// TIA Portal project "XC221" (V12)

(* hardware
DEVICE "S7-1200 station_1"  SIMATIC 1200-Station
   slot 0: "S7-1200 rack"  Rack  V1.0
   slot 1: "PLC_123"  CPU 1214C DC/DC/DC  6ES7 214-1AG31-0XB0  V3.0
   slot 3: "AQ1 x 12 bits"  6ES7 232-4HA30-0XB0  V1.0
*)

// ===== PLC "PLC_123"  CPU 1214C DC/DC/DC =====
// protected blocks, not shown: "EASYPI", "MEMRST"

VAR_GLOBAL   // PLC tag table "Default tag table"
   "System_Byte" AT %MB1 : Byte;
   "FirstScan" AT %M1.0 : Bool;
   "DiagStatusUpdate" AT %M1.1 : Bool;
   "AlwaysTRUE" AT %M1.2 : Bool;
   "AlwaysFALSE" AT %M1.3 : Bool;
   "Clock_Byte" AT %MB0 : Byte;
   "Clock_10Hz" AT %M0.0 : Bool;
   "Clock_5Hz" AT %M0.1 : Bool;
   "Clock_2.5Hz" AT %M0.2 : Bool;
   "Clock_2Hz" AT %M0.3 : Bool;
   "Clock_1.25Hz" AT %M0.4 : Bool;
   "Clock_1Hz" AT %M0.5 : Bool;
   "Clock_0.625Hz" AT %M0.6 : Bool;
   "Clock_0.5Hz" AT %M0.7 : Bool;
END_VAR

VAR_GLOBAL   // PLC tag table "11 - Parâmetros"
   "Par_VT101_HorLim" AT %MD705 : Real;   // Limite de Horas do Ventilador 1
   "Par_VT102_HorLim" AT %MD709 : Real;   // Limite de Horas do Ventilador 2
   "Par_LT101_LimHH" AT %MD713 : Real;   // Limite para a condição “Muito Alto” [mm]
   "Par_LT101_LimH" AT %MD717 : Real;   // Limite para a condição “Alto” [mm]
   "Par_LT101_LimL" AT %MD721 : Real;   // Limite para a condição “Baixo" [mm]
   "Par_LT101_LimLL" AT %MD725 : Real;   // Limite para a condição “Muito Baixo” [mm]
   "Par_LT101_LimDsg" AT %MD729 : Real;   // Limite para desligar a bomba[mm]
   "Par_LT101_LimLig" AT %MD733 : Real;   // Limite para ligar a bomba [mm]
   "Par_LC102_SetPoint" AT %MD737 : Real;   // Setpoint [mm]
   "Par_LC102_Prop" AT %MD741 : Real;   // Ganho proporcional
   "Par_LC102_Integ" AT %MD745 : Real;   // Ganho integral [segundos]
   "Par_BA101_HorLim" AT %MD753 : Real;   // Limite de horas da bomba
   "Par_BA101_RefVel" AT %MD757 : Real;   // Referência de velocidade da bomba [%]
END_VAR

VAR_GLOBAL   // PLC tag table "10 - Analógicas"
   "Ana_GERAL_AtvCPU" AT %MD601 : Real;   // Sinalizador de atividade da CPU
   "Ana_VT101_HorDec" AT %MD605 : Real;   // Horas restantes do ventilador 1
   "Ana_VT102]_HorDec" AT %MD609 : Real;   // Horas restantes do ventilador 2
   "Ana_LT101_Nivel" AT %MD613 : Real;   // Nível de água no tanque [mm]
   "Ana_LC102_SinCtrl" AT %MD617 : Real;   // Sinal de controle [%]
   "Ana_BA101_HorDec" AT %MD621 : Real;   // Horas restantes da bomba
   "Ana_BA101_VelBmb" AT %MD625 : Real;   // Velocidade atual da bomba [%]
END_VAR

VAR_GLOBAL   // PLC tag table "09 - Auxiliares Analógicos"
   "AAu_VT101_Horas" AT %MD505 : Real;   // Horas trabalhadas do ventilador 1
   "AAu_VT101_Minutos" AT %MD509 : Real;   // Minutos trabalhados do ventilador 1
   "AAu_VT101_Segs" AT %MD513 : Real;   // Segundos trabalhados do ventilador 1
   "AAu_VT102_Horas" AT %MD517 : Real;   // Horas trabalhadas do ventilador 2
   "AAu_VT102_Minutos" AT %MD521 : Real;   // Minutos trabalhados do ventilador 2
   "AAu_VT102_Segs" AT %MD525 : Real;   // Segundos trabalhados do ventilador 2
   "AAu_LT101_NivelFP" AT %MD533 : Real;   // Nível em formato real [bruto]
   "AAu_LC102_LstErr" AT %MD553 : Real;   // Último valor de erro
   "AAu_LC102_LstInt" AT %MD557 : Real;   // Último valor da ação integral
   "AAu BA101 Horas" AT %MD537 : Real;   // Horas trabalhadas da bomba
   "AAu BA101 Minutos" AT %MD541 : Real;   // Minutos trabalhados da bomba
   "AAu BA101 Segs" AT %MD545 : Real;   // Segundos trabalhados da bomba
   "AAu BA101 VelBmb" AT %MD549 : Real;   // Velocidade em formato real [bruto]
END_VAR

VAR_GLOBAL   // PLC tag table "08 - Auxiliares Digitais"
   "DAu_GERAL_Rearma" AT %M401.0 : Bool;   // Algum botão de rearme atuado
   "DAu_GERAL_Pul1s0" AT %M401.1 : Bool;   // Pulso de 1 scan a cada 1.0 segundo
   "DAu_VS101_AbrLoc" AT %M402.0 : Bool;   // Abre via modo local
   "DAu_VS101_AbrRem" AT %M402.1 : Bool;   // Abre via modo remoto
   "DAu_VT101_LigLoc" AT %M403.0 : Bool;   // Liga via modo local
   "DAu_VT101_LigRem" AT %M403.1 : Bool;   // Liga via modo remoto
   "DAu_VT101_EdgLig" AT %M403.2 : Bool;   // Borda para ligar ventilador 1
   "DAu_VT101_EdgDsg" AT %M403.3 : Bool;   // Borda para desligar ventilador 1
   "DAu_VT102_LigLoc" AT %M404.0 : Bool;   // Liga via modo local
   "DAu_VT102_LigRem" AT %M404.1 : Bool;   // Liga via modo remoto
   "DAu_VT102_EdgLig" AT %M404.2 : Bool;   // Borda para ligar ventilador 2
   "DAu_VT102_EdgDsg" AT %M404.3 : Bool;   // Borda para desligar ventilador 2
   "DAu_BA101_LigMan" AT %M408.0 : Bool;   // Liga via modo manual
   "DAu_BA101_LigOnOff" AT %M408.1 : Bool;   // Liga via modo On/Off
   "DAu_BA101_LigPID" AT %M408.2 : Bool;   // Liga via modo PID
END_VAR

VAR_GLOBAL   // PLC tag table "07 - Alarmes"
   "Alr_GERAL_Emerge" AT %M301.0 : Bool;   // Condição de emergência ativada
   "Alr_VT101_HorFim" AT %M303.0 : Bool;   // Ventilador 1 com horas esgotadas
   "Alr_VT102_HorFim" AT %M304.0 : Bool;   // Ventilador 2 com horas esgotadas
   "Alr_LT101_ExcedHH" AT %M305.0 : Bool;   // Limite “Muito Alto” excedido
   "Alr_LT101_ExcedH" AT %M305.1 : Bool;   // Limite “Alto” excedido
   "Alr_LT101_ExcedL" AT %M305.2 : Bool;   // Limite “Baixo” excedido
   "Alr LT101_ExcedLL" AT %M305.3 : Bool;   // Limite “Muito Baixo” excedido
   "Alr_BA101_HorFim" AT %M308.0 : Bool;   // Bomba com horas esgotadas
   "Alr_BA101_DisjOff" AT %M308.1 : Bool;   // Disjuntor da bomba desarmado
END_VAR

DATA_BLOCK "AUXPRG"   // DB1
TITLE = Variáveis auxiliares para programação
{ S7_Optimized_Access := 'FALSE' }
AUTHOR : Dimitri
VERSION : 0.1
// Posições de memória para uso em temporizadores, contadores, instruções de detecção de borda etc.
   VAR
      "Timer" : Array [1 .. 20] of IEC_TIMER;
      "Counter" : Array [1 .. 20] of IEC_COUNTER;
      Edge : Array [1 .. 20] of Bool;
   END_VAR
BEGIN
END_DATA_BLOCK

ORGANIZATION_BLOCK "Main"   // OB1, LAD, ProgramCycle
TITLE = Ciclo principal do programa
{ S7_Optimized_Access := 'FALSE' }
VERSION : 0.1
BEGIN
END_ORGANIZATION_BLOCK